// TIA Portal V20 export
TYPE "LER_typeGearInMonitoring"
// stored: Access Published
   STRUCT
      startSync : Bool;
      inSync : Bool;
      continuousUpdateActive : Bool;
      busy : Bool;
      commandAborted : Bool;
      error : Bool;
      errorId : Word;
   END_STRUCT;
END_TYPE
